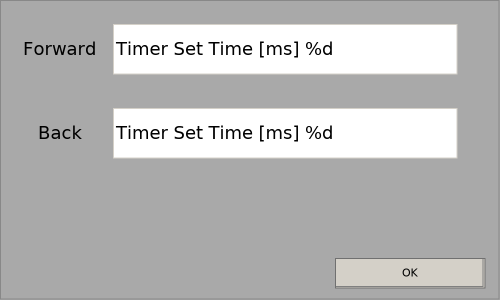
VISUALIZATION DialogTimer_GripperPosi  // 500x300
    Button (335,258 150x30), "OK"
        OnMouseClick: CloseDialog Dialog=DialogTimer_GripperPosi, Result=OK, NumpadKeypadSet=True
    Textfield (113,24 344x50), "Timer Set Time [ms] %d", text variable: PersistentStruct.TimeGripperStartPosition
        OnMouseClick: write the text variable via Edit
    Textfield (113,108 344x50), "Timer Set Time [ms] %d", text variable: PersistentStruct.TimeGripperHomePosition
        OnMouseClick: write the text variable via Edit
    Label (4,34 112x30), "Forward"
    Label (4,118 112x30), "Back"
END_VISUALIZATION

(* stored: Version 1.1.0.1, ProductVersion 3.1.4024.3
   Visu DialogTimer_GripperPosi: Id {226396e7-4baf-43d3-b05b-9559b06e1d3a} *)
